{attribute 'qualified_only'}
TYPE E_EVENTQUALIFIERMODE :
(
	Reserved := 0,
    EventSingleShot := 1,
    EventDisappears := 2,
    EventAppears := 3
) USINT;
END_TYPE

(* stored: Version 1.1.0.1, ProductVersion 3.1.4022.18
   DUT E_EVENTQUALIFIERMODE: Id {812ac71b-e127-44cf-93ca-871b14abbe58} *)
